Staubli VAL3: getStatus.pgx

public program getStatus(num& x_nStatus[] (dimensions=1))
  local num l_nStatus
begin
  // This program returns the status of the encoder librairie
  //
  // Input Param
  // None
  //
  // Output Param
  //  x_nStatus    : Status of the encoder library
  //
  //Created 04-06-07                              C.CURRIVAND
  //--------------------------------------------------------------
  l_nStatus=taskStatus(sTASK)
  switch l_nStatus
    // Task not created (yet !)
    case -1
      x_nStatus=3999
    break
    // Task running
    case 0,1
      x_nStatus=0
    break
    // Run-time error
    default
      x_nStatus=3000+l_nStatus
    break
  endSwitch
end
